SUBAPPLICATION Uebung_055 (* DigitalInput_I1-_I4 auf DigitalOutput_Q1-_Q4 *)
  (* Standard: 61499-2 *)
  (* Version 1.0, 2023-10-23, franz *)
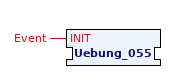
  EVENT_INPUT
    INIT;
  END_EVENT
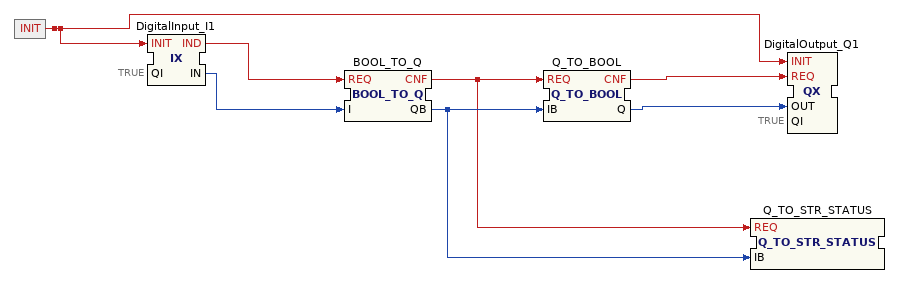
  FBS
    DigitalOutput_Q1 : QX(QI := TRUE);
    DigitalInput_I1 : IX(QI := TRUE);
    BOOL_TO_Q : BOOL_TO_Q;
    Q_TO_BOOL : Q_TO_BOOL;
    Q_TO_STR_STATUS : Q_TO_STR_STATUS;
  END_FBS
  EVENT_CONNECTIONS
    INIT TO DigitalInput_I1.INIT;
    INIT TO DigitalOutput_Q1.INIT;
    BOOL_TO_Q.CNF TO Q_TO_BOOL.REQ;
    Q_TO_BOOL.CNF TO DigitalOutput_Q1.REQ;
    DigitalInput_I1.IND TO BOOL_TO_Q.REQ;
    BOOL_TO_Q.CNF TO Q_TO_STR_STATUS.REQ;
  END_CONNECTIONS
  DATA_CONNECTIONS
    BOOL_TO_Q.QB TO Q_TO_BOOL.IB;
    DigitalInput_I1.IN TO BOOL_TO_Q.I;
    Q_TO_BOOL.Q TO DigitalOutput_Q1.OUT;
    BOOL_TO_Q.QB TO Q_TO_STR_STATUS.IB;
  END_CONNECTIONS
END_SUBAPPLICATION
